// TIA Portal V19 export
ORGANIZATION_BLOCK "Main"   // OB1, LAD, ProgramCycle
TITLE = "Main Program Sweep (Cycle)"
{ S7_Optimized_Access := 'TRUE' }
// stored: SetENOAutomatically false
   VAR_INPUT
      Initial_Call : Bool;   // Initial call of this OB
      Remanence : Bool;   // =True, if remanent data are available
   END_VAR
BEGIN

REGION Network 1
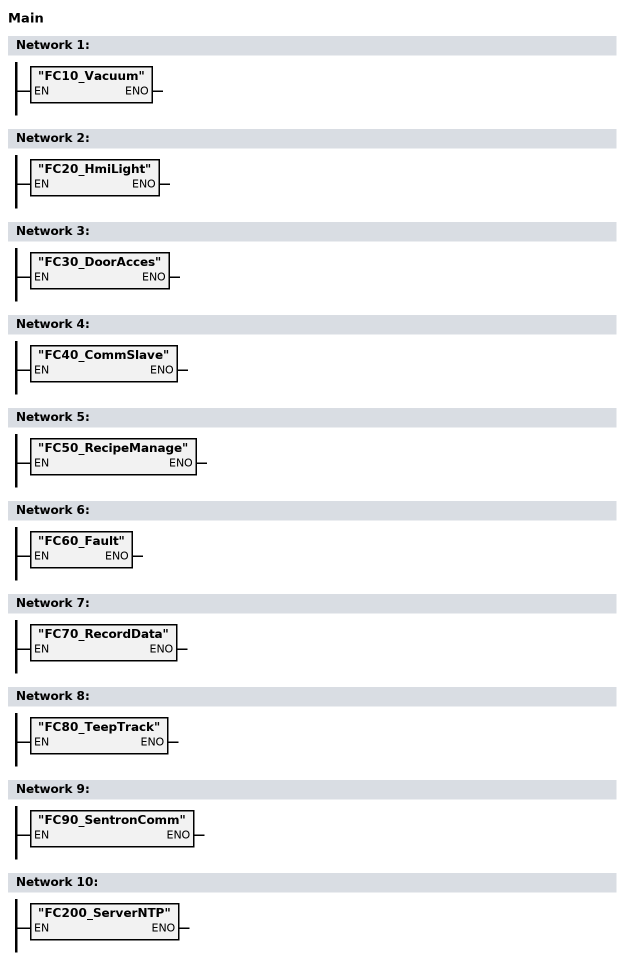
   RUNG wire#powerrail
      "FC10_Vacuum"()
   END_RUNG
   // the same network as SCL:
   "FC10_Vacuum"();
END_REGION

REGION Network 2
   RUNG wire#powerrail
      "FC20_HmiLight"()
   END_RUNG
   // the same network as SCL:
   "FC20_HmiLight"();
END_REGION

REGION Network 3
   RUNG wire#powerrail
      "FC30_DoorAcces"()
   END_RUNG
   // the same network as SCL:
   "FC30_DoorAcces"();
END_REGION

REGION Network 4
   RUNG wire#powerrail
      "FC40_CommSlave"()
   END_RUNG
   // the same network as SCL:
   "FC40_CommSlave"();
END_REGION

REGION Network 5
   RUNG wire#powerrail
      "FC50_RecipeManage"()
   END_RUNG
   // the same network as SCL:
   "FC50_RecipeManage"();
END_REGION

REGION Network 6
   RUNG wire#powerrail
      "FC60_Fault"()
   END_RUNG
   // the same network as SCL:
   "FC60_Fault"();
END_REGION

REGION Network 7
   RUNG wire#powerrail
      "FC70_RecordData"()
   END_RUNG
   // the same network as SCL:
   "FC70_RecordData"();
END_REGION

REGION Network 8
   RUNG wire#powerrail
      "FC80_TeepTrack"()
   END_RUNG
   // the same network as SCL:
   "FC80_TeepTrack"();
END_REGION

REGION Network 9
   RUNG wire#powerrail
      "FC90_SentronComm"()
   END_RUNG
   // the same network as SCL:
   "FC90_SentronComm"();
END_REGION

REGION Network 10
   RUNG wire#powerrail
      "FC200_ServerNTP"()
   END_RUNG
   // the same network as SCL:
   "FC200_ServerNTP"();
END_REGION
END_ORGANIZATION_BLOCK
